PROGRAM task5
VAR
	myTime : TIME := T#10S;
	fbTimeOn : TON := (PT := myTime);
	myBool : BOOL := TRUE;
END_VAR

fbTimeOn(IN := myBool);

END_PROGRAM

(* stored: Version 1.1.0.1, ProductVersion 3.1.4024.12
   POU task5: Id {ccc76bc9-05fc-4160-8aa2-1a4ae11942f4}, SpecialFunc None *)
